// Registers an I_Generic owner in the global entity list.
FUNCTION_BLOCK FINAL Entity IMPLEMENTS I_Entity
VAR
	{attribute 'no_copy'}
	{attribute 'no_init'}
	_iGeneric: I_Generic;	
	_iNext: I_Entity;
	_iPrev: I_Entity;
	_eResult: Result;
END_VAR

PROPERTY INTERNAL _Next : I_Entity
GET
_Next := _iNext;
END_GET
SET
_iNext := _Next;
END_SET
END_PROPERTY

PROPERTY INTERNAL _Prev : I_Entity
GET
_Prev := _iPrev;
END_GET
SET
_iPrev := _Prev;
END_SET
END_PROPERTY

PROPERTY INTERNAL _Raw : I_Generic
GET
_Raw := _iGeneric;
END_GET
SET
_iGeneric := _Raw;
END_SET
END_PROPERTY

PROPERTY INTERNAL _Result : Result
GET
_Result := _eResult;
END_GET
END_PROPERTY

//FB_Exit must be implemented explicitly. If there is an implementation, then the
//method is called before the controller removes the code of the function block instance
//(implicit call). The return value is not evaluated.
{attribute 'hide'}
METHOD FB_Exit: BOOL
VAR_INPUT
    bInCopyCode: BOOL;  // TRUE: the exit method is called in order to leave the instance which will be copied afterwards (online change).  
END_VAR
IF NOT bInCopyCode THEN
	IF Plant._DetachEntity(THIS^) = Ok THEN
		_Plant.bOnlineChangeEntityDeleted := TRUE;
	END_IF
END_IF
END_METHOD

// Registers iGeneric during initialization; panics if iGeneric is 0.
{attribute 'hide'}
METHOD FB_Init: BOOL
VAR_INPUT
    bInitRetains: BOOL; // TRUE on retain initialization.
    bInCopyCode: BOOL;  // TRUE before online-change copy.
	iGeneric: I_Generic; // Owner to register; must not be 0.
END_VAR
IF iGeneric = 0 THEN
	_eResult := Error;
	Plant.Panic(THIS^, 'Entity cannot be initialized with 0');
	RETURN;

END_IF

_iGeneric := iGeneric;

IF _eResult <> None THEN
	RETURN;
END_IF

IF (_eResult := Plant._AttachEntity(THIS^)) = Ok THEN
	_Plant.bOnlineChangeEntityCreated := TRUE;
ELSE
	Plant.Panic(THIS^, __POUNAME());
END_IF
END_METHOD

// Raw discoverable interface for __QUERYINTERFACE.
PROPERTY Raw : I_Generic
GET
Raw := _iGeneric;
END_GET
END_PROPERTY

{attribute 'hide'}
METHOD ValidateInterface
END_METHOD

END_FUNCTION_BLOCK

(* stored: Version 1.1.0.1
   POU Entity: Id {a874bde5-f689-48f5-96c9-83b47d2bb01b}, SpecialFunc None
   Property _Next: Id {8d0df887-d92e-47e4-9173-d51dc5f71061}
   Get Get: Id {69c479c6-496d-4544-8e03-2fa101a500bd}
   Set Set: Id {1d587535-a01f-42f1-90a8-6913adb4690d}
   Property _Prev: Id {dc959834-2b1f-412a-84d1-9286f005eb2d}
   Get Get: Id {a91a7dde-6ccb-4e09-ba88-706222add5e4}
   Set Set: Id {d3db405a-7139-4c8d-84b4-96f56835e7f4}
   Property _Raw: Id {84bc605e-077c-4e23-bbd5-93ce370af17c}
   Get Get: Id {7c364d4d-4000-47ec-b72c-702748352337}
   Set Set: Id {995e244f-c388-41a4-ac14-937884337efd}
   Property _Result: Id {32a97810-b8fd-4467-843e-b19132c8f3f4}
   Get Get: Id {636a706b-3bf6-496c-89d6-d262add3263b}
   Method FB_Exit: Id {42208c5b-7f6e-464d-8c2a-eeb37816f581}
   Method FB_Init: Id {30a5db3d-56de-4ed6-bc93-41367e567754}
   Property Raw: Id {80501f44-2696-4f4b-ba62-8e5556db4eab}
   Get Get: Id {3d5d7f86-a929-4c23-81d0-7c6ff884abb3}
   Method ValidateInterface: Id {e34bd26f-f29f-49cc-8f20-b10bb8bf4181} *)
